TYPE DigitalOutputBase_1FE0D5EE :
STRUCT
END_STRUCT
END_TYPE

(* stored: Version 1.2.0.0, ProductVersion 3.1.4024.9
   DUT DigitalOutputBase_1FE0D5EE: Id {62b58711-f9ac-421b-b953-81124387923b} *)
